(* PLC project Example for PtP Library, CODESYS CODESYS V3.5 SP22 Patch 1, author chmm *)
(* stored: creationDateTime 2026-05-20T11:17:28.3006532, version 3.5.0.11, modificationDateTime 2025-11-25T04:17:57, organization Festo AG & Co. KG *)

PROGRAM PLC_PRG
  VAR
    ActPos : REAL;
    ActVelo : REAL;
    ActTorq : REAL;
    Power_CMMT : MC_Power_Festo;
    Reset_CMMT : MC_Reset_Festo;
    Home_CMMT : MC_Home_Festo;
    Halt_CMMT : MC_Halt_Festo;
    MoveAbs_CMMT : MC_MoveAbsolute_Festo;
    MoveRel_CMMT : MC_MoveRelative_Festo;
    ReadParam_CMMT : MC_ReadParameter_Festo;
    WriteParam_CMMT : MC_WriteParameter_Festo;
    ReadPos_CMMT : MC_ReadActualPosition_Festo;
    ReadTorq_CMMT : MC_ReadActualTorque_Festo;
    ReadVelo_CMMT : MC_ReadActualVelocity_Festo;
    ReadStatus_CMMT : MC_ReadStatus_Festo;
    ReadAxisErr_CMMT : MC_ReadAxisError_Festo;
    MoveAdd_CMMT : MC_MoveAdditive_Festo;
    Stop_CMMT : MC_Stop_Festo;
    MoveVelo_CMMT : MC_MoveVelocity_Festo;
    TorqControl_CMMT : MC_TorqueControl_Festo;
    Jog_CMMT : MC_Jog_Festo;
    Record_CMMT : MC_RecordTable_Festo;
    ReadStringParam_CMMT : MC_ReadStringParameter_Festo;
    WriteStringParam_CMMT : MC_WriteStringParameter_Festo;
    ReadAxisInfo_CMMT : MC_ReadAxisInfo_Festo;
    DeviceService_CMMT : MC_DeviceService_Festo;
  END_VAR

                    ActPos			:= CMMT_AS_MP_S1.ActualPosition;
ActVelo			:= CMMT_AS_MP_S1.ActualVelocity;
ActTorq			:= CMMT_AS_MP_S1.ActualTorque;

Power_CMMT(Axis:=CMMT_AS_MP_S1);
Reset_CMMT(Axis:=CMMT_AS_MP_S1);
Home_CMMT(Axis:=CMMT_AS_MP_S1);
Halt_CMMT(Axis:=CMMT_AS_MP_S1);
MoveAbs_CMMT(Axis:=CMMT_AS_MP_S1);
MoveRel_CMMT(Axis:=CMMT_AS_MP_S1);
ReadParam_CMMT(Axis:=CMMT_AS_MP_S1);
WriteParam_CMMT(Axis:=CMMT_AS_MP_S1);
ReadPos_CMMT(Axis:=CMMT_AS_MP_S1);
ReadTorq_CMMT(Axis:=CMMT_AS_MP_S1);
ReadVelo_CMMT(Axis:=CMMT_AS_MP_S1);
ReadStatus_CMMT(Axis:=CMMT_AS_MP_S1);
ReadAxisErr_CMMT(Axis:=CMMT_AS_MP_S1);
MoveAdd_CMMT(Axis:=CMMT_AS_MP_S1);
Stop_CMMT(Axis:=CMMT_AS_MP_S1);
MoveVelo_CMMT(Axis:=CMMT_AS_MP_S1);
TorqControl_CMMT(Axis:=CMMT_AS_MP_S1);
Jog_CMMT(Axis:=CMMT_AS_MP_S1);
Record_CMMT(Axis:=CMMT_AS_MP_S1);
ReadStringParam_CMMT(Axis:=CMMT_AS_MP_S1);
WriteStringParam_CMMT(Axis:=CMMT_AS_MP_S1);
ReadAxisInfo_CMMT(Axis:=CMMT_AS_MP_S1);
DeviceService_CMMT(Axis:=CMMT_AS_MP_S1);
                  
END_PROGRAM

CONFIGURATION Device
  RESOURCE Application ON PLC
    TASK MainTask(INTERVAL := T#2ms, PRIORITY := 1);
    TASK EtherCAT_Task(INTERVAL := T#2ms, PRIORITY := 1);
    PROGRAM PLC_PRG WITH MainTask : PLC_PRG;
  END_RESOURCE
END_CONFIGURATION

CONFIGURATION SPS_Diagnose
END_CONFIGURATION

CONFIGURATION CPX_E_System
END_CONFIGURATION

CONFIGURATION E_CEC_M1_PN
END_CONFIGURATION

CONFIGURATION EtherCAT_Master
END_CONFIGURATION

CONFIGURATION CMMT_AS_MP_S1
END_CONFIGURATION

CONFIGURATION PROFINET_Device
END_CONFIGURATION

CONFIGURATION SoftMotion General Axis Pool
END_CONFIGURATION
